(* IEC 61131-3 sources: Std_PalletMover/Class/Wewo_EnumBase, 1 file *)

(* ---- Wewo_EnumBase.st ---- *)
(*!
<Class
	Name               = "Wewo_EnumBase"
	Revision           = "0.0"
	RealtimeTask       = "false"
	CyclicTask         = "false"
	BackgroundTask     = "false"
	Sigmatek           = "false"
	OSInterface        = "false"
	HighPriority       = "false"
	Automatic          = "false"
	UpdateMode         = "Prescan"
	SharedCommandTable = "true"
	Objectsize         = "(654,120)"
	Comment            = "reference table for enum variables.&#13;&#10;&#13;&#10;ObjectName is used to translate objectId into variablename string&#13;&#10;&#13;&#10;Server columnIdx:  Select which column should be used to write enum text&#13;&#10;">
	<Channels>
		<Server Name="columnIdx" Visualized="false" Initialize="true" DefValue="0" WriteProtected="false" Retentive="false" Comment="Select which column should be used to write enum text&#13;&#10;idx = -1 Value not written&#13;&#10;idx &gt;=0  write value"/>
	</Channels>
	<Network Name="Wewo_EnumBase">
		<!-- List of Components in this network -->
		<Components>
			<Object
				Name       = "_base"
				Class      = "Wewo_LinkedObjectBase"
				Position   = "(218,120)"
				Visualized = "false">
				<Channels>
					<Server Name="m_Id"/>
					<Server Name="m_p_Name"/>
					<Server Name="o_ErrorWarningStatus"/>
					<Server Name="ObjectStatus"/>
					<Server Name="ToObject"/>
					<Client Name="c_Group"/>
					<Client Name="op_LogData"/>
					<Client Name="p_NextObject"/>
					<Client Name="p_PreviousObject"/>
				</Channels>
			</Object>
		</Components>
		<Comments>
		</Comments>
		<!-- List of Connections in this network -->
		<Connections>
			<Connection Source="this.ToObject" Destination="_base.ToObject" Vertices="(1060,210),(888,210),"/>
			<Connection Source="this.ObjectStatus" Destination="_base.ObjectStatus" Vertices="(1060,270),(888,270),"/>
			<Connection Source="this.o_ErrorWarningStatus" Destination="_base.o_ErrorWarningStatus" Vertices="(1060,330),(888,330),"/>
			<Connection Source="this.m_Id" Destination="_base.m_Id" Vertices="(1060,390),(888,390),"/>
			<Connection Source="this.m_p_Name" Destination="_base.m_p_Name" Vertices="(1060,450),(888,450),"/>
			<Connection Source="_base.op_LogData" Destination="this.op_LogData" Vertices="(218,210),(38,210),"/>
			<Connection Source="_base.p_NextObject" Destination="this.p_NextObject" Vertices="(218,390),(38,330),"/>
			<Connection Source="_base.c_Group" Destination="this.c_Group" Vertices="(218,270),(38,270),"/>
		</Connections>
		<!-- Headerfiles -->
		<Options>
		</Options>
	</Network>
</Class>
*)
#pragma using Wewo_LinkedObjectBase

Wewo_EnumBase : CLASS
: Wewo_LinkedObjectBase
	TYPE
#pragma pack(push, 1)
	  t_EnumStruct : STRUCT
	    id : DINT;
	    p_String : ^CHAR;
	  END_STRUCT;
#pragma pack(pop)
	END_TYPE
  //Servers:
	columnIdx 	: SvrCh_UDINT;
  //Clients:
  //Variables:
		p_StartOfTable 	: ^t_EnumStruct;
		nrOfEntries 	: UDINT;
  //Functions:

	FUNCTION VIRTUAL GLOBAL Init;

	FUNCTION VIRTUAL InstallEnumTable;

	FUNCTION VIRTUAL SetTableEntry
		VAR_INPUT
			idx 	: UDINT;
			id 	: DINT;
			p_String 	: ^CHAR;
		END_VAR;

	FUNCTION VIRTUAL GLOBAL GetEnumString
		VAR_INPUT
			id 	: DINT;
		END_VAR
		VAR_OUTPUT
			p_String 	: ^CHAR;
		END_VAR;

	FUNCTION GLOBAL GetEnumVarName
		VAR_OUTPUT
			p_name 	: ^CHAR;
		END_VAR;

	FUNCTION VIRTUAL GLOBAL columnIdx::Write
		VAR_INPUT
			input (EAX) 	: UDINT;
		END_VAR
		VAR_OUTPUT
			result (EAX) 	: UDINT;
		END_VAR;
  //Tables:
	FUNCTION @STD
		VAR_OUTPUT
			ret_code	: CONFSTATES;
		END_VAR;
	FUNCTION GLOBAL TAB @CT_;
END_CLASS;

(*
// TextTableROM is inplemented in derived class
FUNCTION TAB Wewo_EnumBase::TextTableROM
// IdNr,            *pString,
   0  $TYPE_IDX0,   "String 0"  $TYPE_IDX1,
   0  $TYPE_IDX0,   NIL         $TYPE_IDX1            // Close Table

END_FUNCTION
*)

FUNCTION VIRTUAL GLOBAL Wewo_EnumBase::Init
  Wewo_LinkedObjectBase::Init();

  if (initCnt >= 12) then
    columnIdx := columnIdx.Read();

    InstallEnumTable();

  end_if;

END_FUNCTION

// InstallEnumTable() Has to be defined/filled in derviced class
FUNCTION VIRTUAL Wewo_EnumBase::InstallEnumTable

  // Init table administration
  p_StartOfTable := NIL;
  nrOfEntries   := 0;

  // Install entries
  // SetTableEntry(idx:=0, id := 0, p_String := "string text");

END_FUNCTION

FUNCTION VIRTUAL Wewo_EnumBase::SetTableEntry
	VAR_INPUT
		idx 	: UDINT;
		id 	: DINT;
		p_String 	: ^CHAR;
	END_VAR

  VAR
  	p_Entry : ^t_EnumStruct;
  END_VAR

  if ( (p_StartOfTable <> NIL) L_AND (idx < nrOfEntries) ) then
    p_Entry           := p_StartOfTable + idx * sizeof(t_EnumStruct);
    p_Entry^.id       := id;
    p_Entry^.p_String := p_String;

  else
    WriteActiveErrorWarning(IntErrorWarningId:=MSGID_INVALID_OBJECT, LogLevel:=LL_ERROR_CRITICAL, p_msg:="Wewo_EnumBase::SetTableEntry");

  end_if;

END_FUNCTION

FUNCTION VIRTUAL GLOBAL Wewo_EnumBase::GetEnumString
	VAR_INPUT
		id 	: DINT;
	END_VAR
	VAR_OUTPUT
		p_String 	: ^CHAR;
	END_VAR

  VAR
  	p_Entry : ^t_EnumStruct;
    idx     : UDINT;

  END_VAR

  p_String := NIL;                          // Default nothing found

  if (p_StartOfTable <> NIL) then
    p_Entry := p_StartOfTable;
    idx     := 0;

    while (idx < nrOfEntries) do
      // An entry available
      if (p_Entry^.id = id) then
        // match found
        p_String :=  p_Entry^.p_String;       // Set return value

        exit;                                 // Exit loop

      end_if;

      // Next extry
      idx += 1;
      p_Entry := (p_StartOfTable$UDINT + (idx*sizeof(t_EnumStruct))$UDINT)$^t_EnumStruct;

    end_while;

  end_if;

END_FUNCTION

FUNCTION GLOBAL Wewo_EnumBase::GetEnumVarName
	VAR_OUTPUT
		p_name 	: ^CHAR;
	END_VAR

  p_name := m_p_Name;

END_FUNCTION

FUNCTION VIRTUAL GLOBAL Wewo_EnumBase::columnIdx::Write
	VAR_INPUT
		input (EAX) 	: UDINT;
	END_VAR
	VAR_OUTPUT
		result (EAX) 	: UDINT;
	END_VAR

	columnIdx := input;
 	result := columnIdx;

END_FUNCTION
